{attribute 'qualified_only'}
{attribute 'strict'}
TYPE Dimension : 
(
	X := 0,
	Y := 1,
	Z := 2
)UINT;
END_TYPE

(* stored: Version 1.1.0.1, ProductVersion 3.1.4024.9
   DUT Dimension: Id {87d2bf5d-2e59-0548-0778-2459400fde38} *)
